PROGRAM Ax_01_AxisMoveTypeSelect_02
VAR
	HMI_Motion: FB_HMI_Control;


	tMessageOffset: UINT;
	tNumMessagesPerRow: UINT;
	
	
	MyAdvanceInterlock: BOOL;
	MyReturnInterlock: BOOL;
	
	MyAutoAdvanceCondition: BOOL;
	MyAutoReturnCondition: BOOL;
	
	myAdvancePrompt: BOOL;
	myReturnPrompt: BOOL;
	

	NotUsed: UINT;
	
	gMoveIsAbs: BOOL;
	gMoveIsRel: BOOL;
	isAxisMoving: BOOL;

END_VAR
VAR // added by the converter: edge detectors and wires of the graphical bodies
    _rt1, _rt2, _rt3, _rt4 : R_TRIG;
END_VAR

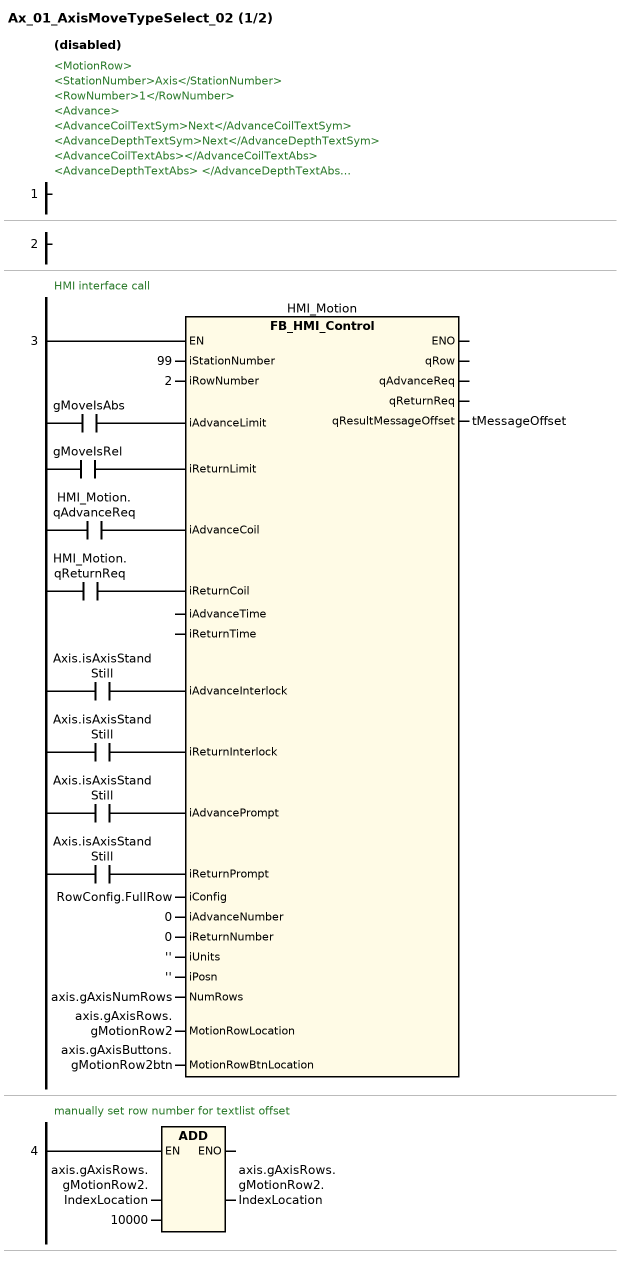
// NETWORK 1 (disabled)
// <MotionRow>
// <StationNumber>Axis</StationNumber>
// <RowNumber>1</RowNumber>
//   <Advance>
//     <AdvanceCoilTextSym>Next</AdvanceCoilTextSym>
//     <AdvanceDepthTextSym>Next</AdvanceDepthTextSym>
//     <AdvanceCoilTextAbs></AdvanceCoilTextAbs>
//     <AdvanceDepthTextAbs> </AdvanceDepthTextAbs>
//     <ManSeq></ManSeq>
//   </Advance>
//   <Return>
//     <ReturnCoilTextSym>Previous</ReturnCoilTextSym>
//     <ReturnDepthTextSym>Previous</ReturnDepthTextSym>
//     <ReturnCoilTextAbs></ReturnCoilTextAbs>
//     <ReturnDepthTextAbs></ReturnDepthTextAbs>
//    <ManSeq></ManSeq>
//   </Return>
//   <Motion>
//     <NameSym>Axis Name</NameSym>
//     <NameAbs>X1</NameAbs>
//   </Motion>
// </MotionRow>

// NETWORK 2

// NETWORK 3
// HMI interface call
HMI_Motion(
    iStationNumber := 99,
    iRowNumber := 2,
    iAdvanceLimit := gMoveIsAbs,
    iReturnLimit := gMoveIsRel,
    iAdvanceCoil := HMI_Motion.qAdvanceReq,
    iReturnCoil := HMI_Motion.qReturnReq,
    iAdvanceInterlock := Axis.isAxisStandStill,
    iReturnInterlock := Axis.isAxisStandStill,
    iAdvancePrompt := Axis.isAxisStandStill,
    iReturnPrompt := Axis.isAxisStandStill,
    iConfig := RowConfig.FullRow,
    iAdvanceNumber := 0,
    iReturnNumber := 0,
    iUnits := '',
    iPosn := '',
    NumRows := axis.gAxisNumRows,
    MotionRowLocation := axis.gAxisRows.gMotionRow2,
    MotionRowBtnLocation := axis.gAxisButtons.gMotionRow2btn,
    qResultMessageOffset => tMessageOffset); // FB_HMI_Control

// NETWORK 4
// manually set row number for textlist offset
axis.gAxisRows.gMotionRow2.IndexLocation := axis.gAxisRows.gMotionRow2.IndexLocation + 10000;

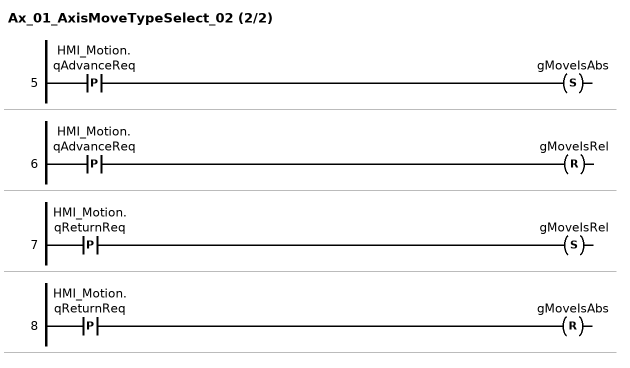
// NETWORK 5
_rt1(CLK := HMI_Motion.qAdvanceReq);
gMoveIsAbs S= _rt1.Q;

// NETWORK 6
_rt2(CLK := HMI_Motion.qAdvanceReq);
gMoveIsRel R= _rt2.Q;

// NETWORK 7
_rt3(CLK := HMI_Motion.qReturnReq);
gMoveIsRel S= _rt3.Q;

// NETWORK 8
_rt4(CLK := HMI_Motion.qReturnReq);
gMoveIsAbs R= _rt4.Q;

END_PROGRAM

(* stored: Version 1.1.0.1, ProductVersion 3.1.4024.12
   POU Ax_01_AxisMoveTypeSelect_02: Id {193668af-76f6-42c2-8f7d-eb8927314956}, SpecialFunc None *)
